TYPE ST_CommunicationConfig :
STRUCT
	sIPAdress: STRING;
	Port: UINT;
	
END_STRUCT
END_TYPE

(* stored: Version 1.1.0.1, ProductVersion 3.1.4026.18
   DUT ST_CommunicationConfig: Id {30496dbe-ef77-43fa-a92a-f084f7770640} *)
